{attribute 'GeneratedUsingTerminal: EK1100-0000-0018'}
{attribute addProperty BoxType "EK1100-0000-0018"}
{attribute addProperty Id "R7_A2_EC_EK1122R7_A2_EC_EK1122_B7F046E468R7_A3_DI_EL1809EL1809_32157CFD20R7_A4_DI_EL1809EL1809_32157CFD20R7_A5_DI_EL1809EL1809_32157CFD20R7_A6_DI_EL1809EL1809_32157CFD20R7_A7_DI_EL1809EL1809_32157CFD20R7_A8_DI_EL1809EL1809_32157CFD20R7_A9_DI_EL1809EL1809_32157CFD20R7_A10_DI_EL1809EL1809_32157CFD20R7_A11_DI_EL1809EL1809_32157CFD20R7_A12_DI_EL1809EL1809_32157CFD20R7_A13_DI_EL2809EL2809_2B6483BD19R7_A14_DI_EL2809EL2809_2B6483BD19R7_EndTerminal_EL9011EL9011_D65D3D320"}
{attribute addProperty CRC "4111325896"}
{attribute addProperty Size "306"}
{attribute addProperty Name "R7 (EK1100)"}
TYPE R7_EK1100_F50DDAC8 EXTENDS EK1100_1FC0878B :
STRUCT
	{attribute addProperty Name "R7_A2_EC (EK1122)"}
	{attribute addProperty PreviousPort "R7 (EK1100) : B"}
	R7_A2_EC_EK1122 : R7_A2_EC_EK1122_B7F046E4;
	{attribute addProperty Name "R7_A3_DI (EL1809)"}
	{attribute addProperty PreviousPort "R7_A2_EC (EK1122) : C"}
	R7_A3_DI_EL1809 : EL1809_32157CFD;
	{attribute addProperty Name "R7_A4_DI (EL1809)"}
	{attribute addProperty PreviousPort "R7_A3_DI (EL1809) : B"}
	R7_A4_DI_EL1809 : EL1809_32157CFD;
	{attribute addProperty Name "R7_A5_DI (EL1809)"}
	{attribute addProperty PreviousPort "R7_A4_DI (EL1809) : B"}
	R7_A5_DI_EL1809 : EL1809_32157CFD;
	{attribute addProperty Name "R7_A6_DI (EL1809)"}
	{attribute addProperty PreviousPort "R7_A5_DI (EL1809) : B"}
	R7_A6_DI_EL1809 : EL1809_32157CFD;
	{attribute addProperty Name "R7_A7_DI (EL1809)"}
	{attribute addProperty PreviousPort "R7_A6_DI (EL1809) : B"}
	R7_A7_DI_EL1809 : EL1809_32157CFD;
	{attribute addProperty Name "R7_A8_DI (EL1809)"}
	{attribute addProperty PreviousPort "R7_A7_DI (EL1809) : B"}
	R7_A8_DI_EL1809 : EL1809_32157CFD;
	{attribute addProperty Name "R7_A9_DI (EL1809)"}
	{attribute addProperty PreviousPort "R7_A8_DI (EL1809) : B"}
	R7_A9_DI_EL1809 : EL1809_32157CFD;
	{attribute addProperty Name "R7_A10_DI (EL1809)"}
	{attribute addProperty PreviousPort "R7_A9_DI (EL1809) : B"}
	R7_A10_DI_EL1809 : EL1809_32157CFD;
	{attribute addProperty Name "R7_A11_DI (EL1809)"}
	{attribute addProperty PreviousPort "R7_A10_DI (EL1809) : B"}
	R7_A11_DI_EL1809 : EL1809_32157CFD;
	{attribute addProperty Name "R7_A12_DI (EL1809)"}
	{attribute addProperty PreviousPort "R7_A11_DI (EL1809) : B"}
	R7_A12_DI_EL1809 : EL1809_32157CFD;
	{attribute addProperty Name "R7_A13_DI (EL2809)"}
	{attribute addProperty PreviousPort "R7_A12_DI (EL1809) : B"}
	R7_A13_DI_EL2809 : EL2809_2B6483BD;
	{attribute addProperty Name "R7_A14_DI (EL2809)"}
	{attribute addProperty PreviousPort "R7_A13_DI (EL2809) : B"}
	R7_A14_DI_EL2809 : EL2809_2B6483BD;
	{attribute addProperty Name "R7_EndTerminal (EL9011)"}
	{attribute addProperty PreviousPort "R7_A14_DI (EL2809) : B"}
	R7_EndTerminal_EL9011 : EL9011_D65D3D32;
END_STRUCT
END_TYPE

(* stored: Version 1.2.0.0, ProductVersion 3.1.4024.11
   DUT R7_EK1100_F50DDAC8: Id {b539b3f1-b000-0c3a-202b-adfd12709965} *)
